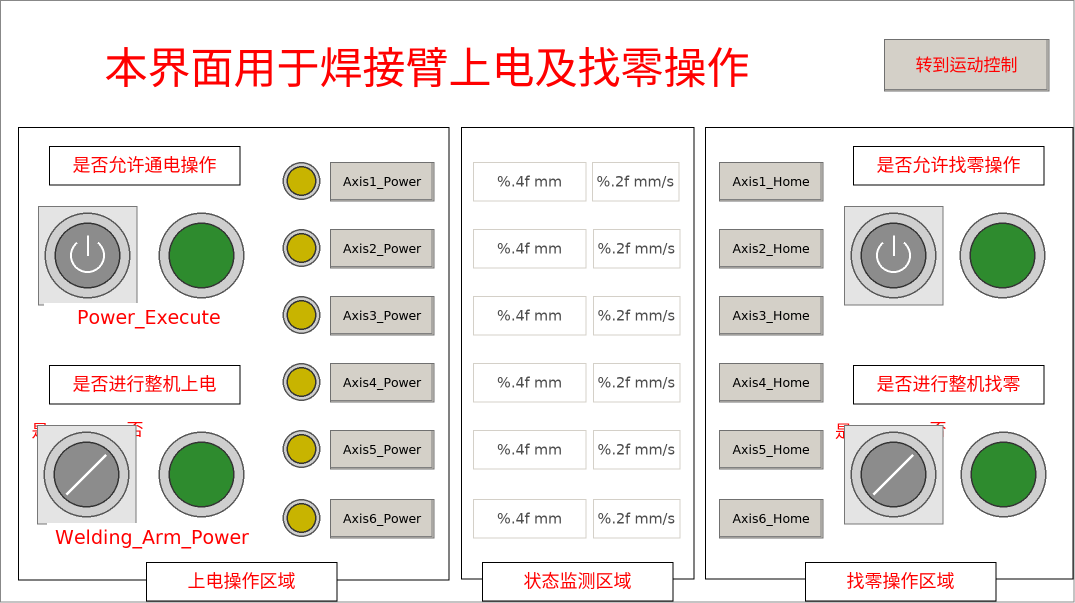
VISUALIZATION Visu_Welding_Arm_Power  // 1075x603
    Rectangle (705,127 368x452)
    Rectangle (461,127 233x452)
    Rectangle (18,127 431x453)
    Label (26,34 802x69), "本界面用于焊接臂上电及找零操作"
    Label (10,416 60x30), "是"
    RoundedRectangle (49,365 191x39), "是否进行整机上电"
    Label (108,416 54x27), "否"
    RoundedRectangle (49,146 191x39), "是否允许通电操作"
    Lamp1 (152,205 99x101), variable: Welding_Arm_Control.Power_Execute, style: Lamp-Lamp1-Green
    PowerSwitch (38,205 99x101), variable: Welding_Arm_Control.Power_Execute, behaviour: TOGGLE, style: Switch-PowerSwitch-Gray
    Lamp1 (152,424 99x101), variable: Welding_Arm_Control.Welding_Arm_Power, style: Lamp-Lamp1-Green
    RotarySwitch (37,424 99x101), variable: Welding_Arm_Control.Welding_Arm_Power, behaviour: TOGGLE, style: Switch-RotarySwitch-Gray
    Label (812,417 63x29), "是"
    RoundedRectangle (853,365 191x39), "是否进行整机找零"
    Label (911,416 54x27), "否"
    RoundedRectangle (853,146 191x39), "是否允许找零操作"
    Lamp1 (953,205 99x101), variable: Welding_Arm_Control.Home_Execute, style: Lamp-Lamp1-Green
    PowerSwitch (844,205 99x101), variable: Welding_Arm_Control.Home_Execute, behaviour: TOGGLE, style: Switch-PowerSwitch-Gray
    Lamp1 (954,424 99x101), variable: Welding_Arm_Control.Welding_Arm_Home_Set, style: Lamp-Lamp1-Green
    RotarySwitch (844,424 99x101), variable: Welding_Arm_Control.Welding_Arm_Home_Set, behaviour: TOGGLE, style: Switch-RotarySwitch-Gray
    Button (884,39 165x52), "转到运动控制"
        OnMouseClick: change screen: Visu_Welding_Arm_SimulinkMove
    Lamp1 (274,159 55x44), variable: Welding_Arm_Control.Power_Status[1], style: Lamp-Lamp1-Yellow
    Button (330,162 104x39), "Axis1_Power"
        toggle Welding_Arm_Control.Axis_Power[1]
    Button (719,162 104x39), "Axis1_Home"
        toggle Welding_Arm_Control.Axis_Home_Set[1]
    Textfield (473,162 113x39), "%.4f mm", text variable: Welding_Arm_Control.Axis_ActPostion[1]
    Textfield (592,162 87x39), "%.2f mm/s", text variable: Welding_Arm_Control.Axis_ActVelocity[1]
    Lamp1 (274,226 55x44), variable: Welding_Arm_Control.Power_Status[2], style: Lamp-Lamp1-Yellow
    Button (330,229 104x39), "Axis2_Power"
        toggle Welding_Arm_Control.Axis_Power[2]
    Button (719,229 104x39), "Axis2_Home"
        toggle Welding_Arm_Control.Axis_Home_Set[2]
    Textfield (473,229 113x39), "%.4f mm", text variable: Welding_Arm_Control.Axis_ActPostion[2]
    Textfield (593,229 87x39), "%.2f mm/s", text variable: Welding_Arm_Control.Axis_ActVelocity[2]
    Lamp1 (274,293 55x44), variable: Welding_Arm_Control.Power_Status[3], style: Lamp-Lamp1-Yellow
    Button (330,296 104x39), "Axis3_Power"
        toggle Welding_Arm_Control.Axis_Power[3]
    Button (719,296 104x39), "Axis3_Home"
        toggle Welding_Arm_Control.Axis_Home_Set[3]
    Textfield (473,296 113x39), "%.4f mm", text variable: Welding_Arm_Control.Axis_ActPostion[3]
    Textfield (593,296 87x39), "%.2f mm/s", text variable: Welding_Arm_Control.Axis_ActVelocity[3]
    Lamp1 (274,360 55x44), variable: Welding_Arm_Control.Power_Status[4], style: Lamp-Lamp1-Yellow
    Button (330,363 104x39), "Axis4_Power"
        toggle Welding_Arm_Control.Axis_Power[4]
    Button (719,363 104x39), "Axis4_Home"
        toggle Welding_Arm_Control.Axis_Home_Set[4]
    Textfield (473,363 113x39), "%.4f mm", text variable: Welding_Arm_Control.Axis_ActPostion[4]
    Textfield (593,363 87x39), "%.2f mm/s", text variable: Welding_Arm_Control.Axis_ActVelocity[4]
    Lamp1 (274,427 55x44), variable: Welding_Arm_Control.Power_Status[5], style: Lamp-Lamp1-Yellow
    Button (330,430 104x39), "Axis5_Power"
        toggle Welding_Arm_Control.Axis_Power[5]
    Button (719,430 104x39), "Axis5_Home"
        toggle Welding_Arm_Control.Axis_Home_Set[5]
    Textfield (473,430 113x39), "%.4f mm", text variable: Welding_Arm_Control.Axis_ActPostion[5]
    Textfield (593,430 87x39), "%.2f mm/s", text variable: Welding_Arm_Control.Axis_ActVelocity[5]
    Lamp1 (274,496 55x44), variable: Welding_Arm_Control.Power_Status[6], style: Lamp-Lamp1-Yellow
    Button (330,499 104x39), "Axis6_Power"
        toggle Welding_Arm_Control.Axis_Power[6]
    Button (719,499 104x39), "Axis6_Home"
        toggle Welding_Arm_Control.Axis_Home_Set[6]
    Textfield (473,499 113x39), "%.4f mm", text variable: Welding_Arm_Control.Axis_ActPostion[6]
    Textfield (593,499 87x39), "%.2f mm/s", text variable: Welding_Arm_Control.Axis_ActVelocity[6]
    RoundedRectangle (146,562 191x39), "上电操作区域"
    RoundedRectangle (482,562 191x39), "状态监测区域"
    Rectangle (44,303 210x29), "Power_Execute"
    Rectangle (47,523 210x29), "Welding_Arm_Power"
    RoundedRectangle (805,562 191x39), "找零操作区域"
END_VISUALIZATION

(* stored: Version 1.1.0.1, ProductVersion 3.1.4020.12
   Visu Visu_Welding_Arm_Power: Id {4cf72fe6-1e06-4608-94bc-323c0475dc76} *)
